// TIA Portal V15.1 export
// export: Created 2024-05-17T05:38:29.3000948Z, ExportSetting WithDefaults, DisplayName Totally Integrated Automation Portal, DisplayVersion V15.1 Update 5, DisplayName TIA Portal Openness, DisplayVersion V15.1 Update 5, DisplayName SINAMICS Startdrive Advanced, DisplayVersion V15.1, DisplayName G130, G150, S120, S150, SINAMICS MV, S210, DisplayVersion V15.1, DisplayName G110M, G120, G120C, G120D, G120P, DisplayVersion V15.1, DisplayName STEP 7 Professional, DisplayVersion V15.1 Update 5, DisplayName STEP 7 Safety, DisplayVersion V15.1, DisplayName WinCC Professional, DisplayVersion V15.1 Update 5, DisplayName SIMATIC Visualization Architect, DisplayVersion V15.1
FUNCTION_BLOCK "LETAFuseCPC20PNSub"   // FB1407, SCL
{ S7_Optimized_Access := 'TRUE' }
VERSION : 0.1
// stored: AutoNumber false, IsIECCheckEnabled false, IsRetainMemResEnabled false, MemoryReserve 100, SetENOAutomatically False, UDAEnableTagReadback false
   VAR_INPUT
      I_NewShift { ExternalAccessible := 'False'; ExternalVisible := 'False'; ExternalWritable := 'False'} : Bool;   // NewShift / Morning shift
      I_ReadNomCurr { ExternalAccessible := 'False'; ExternalVisible := 'False'; ExternalWritable := 'False'} : Bool;   // HMI Command - Read nominal current
      I_CancelReadNomCurr { ExternalAccessible := 'False'; ExternalVisible := 'False'; ExternalWritable := 'False'} : Bool;   // HMI Command - Cancel Read nominal current
      C_HWInput { ExternalAccessible := 'False'; ExternalVisible := 'False'; ExternalWritable := 'False'} : HW_IO;   // Slot ID from CPC20PN
      C_Block1_TotalCurrent { ExternalAccessible := 'False'; ExternalVisible := 'False'; ExternalWritable := 'False'} : HW_IO;   // Base Module Slot ID Total Current, 0=not in use.
      C_Block1_StatusControl { ExternalAccessible := 'False'; ExternalVisible := 'False'; ExternalWritable := 'False'} : HW_IO;   // Base Module Slot ID Status / Control, 0=not in use.
      "C_Block1_MeasurementU/I" { ExternalAccessible := 'False'; ExternalVisible := 'False'; ExternalWritable := 'False'} : HW_IO;   // Base Module Slot ID Measurement UI, 0=not in use.
      C_Block2_TotalCurrent { ExternalAccessible := 'False'; ExternalVisible := 'False'; ExternalWritable := 'False'} : HW_IO;   // Extension Module Slot ID Total Current, 0=not in use.
      C_Block2_StatusControl { ExternalAccessible := 'False'; ExternalVisible := 'False'; ExternalWritable := 'False'} : HW_IO;   // Extension Module Slot ID Status / Control, 0=not in use.
      "C_Block2_MeasurementU/I" { ExternalAccessible := 'False'; ExternalVisible := 'False'; ExternalWritable := 'False'} : HW_IO;   // Extension Module Slot ID Measurement UI, 0=not in use.
      C_Config { ExternalAccessible := 'False'; ExternalVisible := 'False'; ExternalWritable := 'False'} : "ETAFuseCPC20PNConfig";   // Config
   END_VAR
   VAR_OUTPUT
      O_StatusCPC20_Bit0 { ExternalAccessible := 'False'; ExternalVisible := 'False'; ExternalWritable := 'False'} : Bool;   // Bit0 = no configuration data available
      O_StatusCPC20_Bit1 { ExternalAccessible := 'False'; ExternalVisible := 'False'; ExternalWritable := 'False'} : Bool;   // Bit1 = invalid configuration data
      O_StatusCPC20_Bit4 { ExternalAccessible := 'False'; ExternalVisible := 'False'; ExternalWritable := 'False'} : Bool;   // Bit4 = command buffer overflow
      O_StatusCPC20_Bit7 { ExternalAccessible := 'False'; ExternalVisible := 'False'; ExternalWritable := 'False'} : Bool;   // Bit7 = no communication with at least one PWR board
      O_StatusCPC20_Bit9 { ExternalAccessible := 'False'; ExternalVisible := 'False'; ExternalWritable := 'False'} : Bool;   // Bit9 = CPC temporary error
      O_StatusCPC20_Bit10 { ExternalAccessible := 'False'; ExternalVisible := 'False'; ExternalWritable := 'False'} : Bool;   // Bit10 = CPC hardware error
      O_ReadNomCurrActive { ExternalAccessible := 'False'; ExternalVisible := 'False'; ExternalWritable := 'False'} : Bool;   // Reading of nominal current is active
      O_ReadNomCurrFuseNr { ExternalAccessible := 'False'; ExternalVisible := 'False'; ExternalWritable := 'False'} : Int;   // Fuse number Reading of nominal current
      O_AlarmReadNomCurr { ExternalAccessible := 'False'; ExternalVisible := 'False'; ExternalWritable := 'False'} : Bool;   // Overtime Reading of nominal current
      O_Block1TotalCurrent { ExternalAccessible := 'False'; ExternalVisible := 'False'; ExternalWritable := 'False'} : Real;   // Total current Block 1
      O_Block2TotalCurrent { ExternalAccessible := 'False'; ExternalVisible := 'False'; ExternalWritable := 'False'} : Real;   // Total current Block 2
   END_VAR
   VAR_IN_OUT
      IO_ETAFuseData : "ETAFuseData";   // ETA fuse status
      H_ETAFuseCPC20PN : "H_ETAFuseCPC20PN";   // Animation
   END_VAR
   VAR
      InitNominalCurrent { ExternalAccessible := 'False'; ExternalVisible := 'False'; ExternalWritable := 'False'} : Bool;   // Read once all Nominal Currents at Startup
      ChannelNumber { ExternalAccessible := 'False'; ExternalVisible := 'False'; ExternalWritable := 'False'} : Int;   // Channel Number
      Block1Size { ExternalAccessible := 'False'; ExternalVisible := 'False'; ExternalWritable := 'False'} : Int;   // Block size
      Block2Size { ExternalAccessible := 'False'; ExternalVisible := 'False'; ExternalWritable := 'False'} : Int;   // Block size
      HardwareID { ExternalAccessible := 'False'; ExternalVisible := 'False'; ExternalWritable := 'False'} : HW_IO;   // HW IO
      i { ExternalAccessible := 'False'; ExternalVisible := 'False'; ExternalWritable := 'False'} : Int;   // Loop Counter
      iCount { ExternalAccessible := 'False'; ExternalVisible := 'False'; ExternalWritable := 'False'} : Int;   // Loop Counter To Go Threw All Channels
      iCalcAddress { ExternalAccessible := 'False'; ExternalVisible := 'False'; ExternalWritable := 'False'} : Int;   // Fuse Adress To Be Calculated
      iCountGet { ExternalAccessible := 'False'; ExternalVisible := 'False'; ExternalWritable := 'False'} : Int;   // Sequence Pointer Get Data
      iCountNominalCurrent { ExternalAccessible := 'False'; ExternalVisible := 'False'; ExternalWritable := 'False'} : Int;   // Loop Counter To Go Threw All Channels
      BuildStatus { ExternalAccessible := 'False'; ExternalVisible := 'False'; ExternalWritable := 'False'} : Word;   // BuildStatus
      iError { ExternalAccessible := 'False'; ExternalVisible := 'False'; ExternalWritable := 'False'} : Int;   // iError
      CalcValue { ExternalAccessible := 'False'; ExternalVisible := 'False'; ExternalWritable := 'False'} : Int;   // CalcValue
      EmptyDataCPC20 { ExternalAccessible := 'False'; ExternalVisible := 'False'; ExternalWritable := 'False'} : Struct   // Empty struct to delete info
         Voltage { ExternalAccessible := 'False'; ExternalVisible := 'False'; ExternalWritable := 'False'} : Real;   // Voltage
         Current { ExternalAccessible := 'False'; ExternalVisible := 'False'; ExternalWritable := 'False'} : Real;   // Current
         NominalCurrent { ExternalAccessible := 'False'; ExternalVisible := 'False'; ExternalWritable := 'False'} : Byte;   // Nominal Current
         Status { ExternalAccessible := 'False'; ExternalVisible := 'False'; ExternalWritable := 'False'} : Byte;   // Status
         Control { ExternalAccessible := 'False'; ExternalVisible := 'False'; ExternalWritable := 'False'} : Byte;   // Control
      END_STRUCT;
      EmptyForHMIFuse { ExternalAccessible := 'False'; ExternalVisible := 'False'; ExternalWritable := 'False'} : Struct   // Empty struct to delete info
         Used { ExternalAccessible := 'False'; ExternalVisible := 'False'; ExternalWritable := 'False'} : Bool;   // Used
         "SwitchOn/OFFOnlyCabinet" { ExternalAccessible := 'False'; ExternalVisible := 'False'; ExternalWritable := 'False'} : Bool;   // Switch On/Off only posible in the cabinet, button on the fuse
         IAnim { ExternalAccessible := 'False'; ExternalVisible := 'False'; ExternalWritable := 'False'} : Word;   // IAnim
         Status { ExternalAccessible := 'False'; ExternalVisible := 'False'; ExternalWritable := 'False'} : Byte;   // Status
         AlarmActive { ExternalAccessible := 'False'; ExternalVisible := 'False'; ExternalWritable := 'False'} : Bool;   // Alarm Active
      END_STRUCT;
      EmptyForHMIChannelInfo { ExternalAccessible := 'False'; ExternalVisible := 'False'; ExternalWritable := 'False'} : Struct   // Empty struct to delete info
         "Name" { ExternalAccessible := 'False'; ExternalVisible := 'False'; ExternalWritable := 'False'} : String[40];   // Fuse name
         Description { ExternalAccessible := 'False'; ExternalVisible := 'False'; ExternalWritable := 'False'} : String[60];   // Description
         Current { ExternalAccessible := 'False'; ExternalVisible := 'False'; ExternalWritable := 'False'} : Real;   // Current
         NominalCurrent { ExternalAccessible := 'False'; ExternalVisible := 'False'; ExternalWritable := 'False'} : Int;   // Nominal Current
      END_STRUCT;
      NonCyclicCommunication { ExternalAccessible := 'False'; ExternalVisible := 'False'; ExternalWritable := 'False'} : Struct   // Non cyclic communication variables
         H_ReadNomCurrTrig { ExternalAccessible := 'False'; ExternalVisible := 'False'; ExternalWritable := 'False'} : Bool;   // HMI button to start reading nominal current
         ReadNomCurrActive { ExternalAccessible := 'False'; ExternalVisible := 'False'; ExternalWritable := 'False'} : Bool;   // Reading of nominal current is active
      END_STRUCT;
      Get { ExternalAccessible := 'False'; ExternalVisible := 'False'; ExternalWritable := 'False'} : Struct   // FB
         bGetData { ExternalAccessible := 'False'; ExternalVisible := 'False'; ExternalWritable := 'False'} : Bool;
         bValid { ExternalAccessible := 'False'; ExternalVisible := 'False'; ExternalWritable := 'False'} : Bool;
         bBusy { ExternalAccessible := 'False'; ExternalVisible := 'False'; ExternalWritable := 'False'} : Bool;
         diIndex { ExternalAccessible := 'False'; ExternalVisible := 'False'; ExternalWritable := 'False'} : DInt;
         uiMlen { ExternalAccessible := 'False'; ExternalVisible := 'False'; ExternalWritable := 'False'} : UInt;
         uilen { ExternalAccessible := 'False'; ExternalVisible := 'False'; ExternalWritable := 'False'} : UInt;
         bError { ExternalAccessible := 'False'; ExternalVisible := 'False'; ExternalWritable := 'False'} : Bool;
         dwState { ExternalAccessible := 'False'; ExternalVisible := 'False'; ExternalWritable := 'False'} : DWord;
         TonError { ExternalAccessible := 'False'; ExternalVisible := 'False'; ExternalWritable := 'False'} : Bool;
         DataByte { ExternalAccessible := 'False'; ExternalVisible := 'False'; ExternalWritable := 'False'} : Array[1..20] of Byte;
      END_STRUCT;
      RDREC_FB { ExternalAccessible := 'False'; ExternalVisible := 'False'; ExternalWritable := 'False'} : RDREC;   // FB
      StatusCPC20 { ExternalAccessible := 'False'; ExternalVisible := 'False'; ExternalWritable := 'False'} : Array[0..1] of Byte;   // Temp
      Current { ExternalAccessible := 'False'; ExternalVisible := 'False'; ExternalWritable := 'False'} : Array[0..1] of Byte;   // Temp
      Status { ExternalAccessible := 'False'; ExternalVisible := 'False'; ExternalWritable := 'False'} : Array[1..32] of Byte;   // Temp
      Control { ExternalAccessible := 'False'; ExternalVisible := 'False'; ExternalWritable := 'False'} : Array[1..32] of Byte;   // Temp
      UI { ExternalAccessible := 'False'; ExternalVisible := 'False'; ExternalWritable := 'False'} : Array[0..130] of Byte;   // Temp
      T_ReadNomCurr { ExternalAccessible := 'False'; ExternalVisible := 'False'; ExternalWritable := 'False'} : TON_TIME;   // Timer
   END_VAR
BEGIN
   (*=================================================================================*)
   (* Init at startup *)
   (*=================================================================================*)
   IF "FirstScan" THEN
       #InitNominalCurrent := True;
   END_IF;

   (*=================================================================================*)
   (* Check number of protectors active *)
   (*=================================================================================*)
   #Block1Size := 0;
   IF #C_Config.Fuse[1].Used THEN
       #Block1Size := 1;
   END_IF;
   IF #C_Config.Fuse[3].Used THEN
       #Block1Size := 2;
   END_IF;
   IF #C_Config.Fuse[5].Used THEN
       #Block1Size := 3;
   END_IF;
   IF #C_Config.Fuse[7].Used THEN
       #Block1Size := 4;
   END_IF;
   IF #C_Config.Fuse[9].Used THEN
       #Block1Size := 5;
   END_IF;
   IF #C_Config.Fuse[11].Used THEN
       #Block1Size := 6;
   END_IF;
   IF #C_Config.Fuse[13].Used THEN
       #Block1Size := 7;
   END_IF;
   IF #C_Config.Fuse[15].Used THEN
       #Block1Size := 8;
   END_IF;
   IF #C_Config.Fuse[17].Used THEN
       #Block1Size := 9;
   END_IF;
   IF #C_Config.Fuse[19].Used THEN
       #Block1Size := 10;
   END_IF;
   IF #C_Config.Fuse[21].Used THEN
       #Block1Size := 11;
   END_IF;
   IF #C_Config.Fuse[23].Used THEN
       #Block1Size := 12;
   END_IF;
   IF #C_Config.Fuse[25].Used THEN
       #Block1Size := 13;
   END_IF;
   IF #C_Config.Fuse[27].Used THEN
       #Block1Size := 14;
   END_IF;
   IF #C_Config.Fuse[29].Used THEN
       #Block1Size := 15;
   END_IF;
   IF #C_Config.Fuse[31].Used THEN
       #Block1Size := 16;
   END_IF;

   #Block2Size := 0;
   IF #C_Config.Fuse[33].Used THEN
       #Block2Size := 1;
   END_IF;
   IF #C_Config.Fuse[35].Used THEN
       #Block2Size :=2;
   END_IF;
   IF #C_Config.Fuse[37].Used THEN
       #Block2Size := 3;
   END_IF;
   IF #C_Config.Fuse[39].Used THEN
       #Block2Size := 4;
   END_IF;
   IF #C_Config.Fuse[41].Used THEN
       #Block2Size := 5;
   END_IF;
   IF #C_Config.Fuse[43].Used THEN
       #Block2Size := 6;
   END_IF;
   IF #C_Config.Fuse[45].Used THEN
       #Block2Size := 7;
   END_IF;
   IF #C_Config.Fuse[47].Used THEN
       #Block2Size := 8;
   END_IF;
   IF #C_Config.Fuse[49].Used THEN
       #Block2Size := 9;
   END_IF;
   IF #C_Config.Fuse[51].Used THEN
       #Block2Size := 10;
   END_IF;
   IF #C_Config.Fuse[53].Used THEN
       #Block2Size := 11;
   END_IF;
   IF #C_Config.Fuse[55].Used THEN
       #Block2Size := 12;
   END_IF;
   IF #C_Config.Fuse[57].Used THEN
       #Block2Size := 13;
   END_IF;
   IF #C_Config.Fuse[59].Used THEN
       #Block2Size := 14;
   END_IF;
   IF #C_Config.Fuse[61].Used THEN
       #Block2Size := 15;
   END_IF;
   IF #C_Config.Fuse[63].Used THEN
       #Block2Size := 16;
   END_IF;

   (*=================================================================================*)
   (* CPC20   ---   Read State *)
   (*=================================================================================*)
   IF #C_HWInput > 0 THEN
       (*Read Data*)
       #iError := DPRD_DAT(LADDR := #C_HWInput, RECORD => #StatusCPC20);
       (*Calculate Value*)
       #BuildStatus := #StatusCPC20[0];
       #BuildStatus := SHL(IN := #BuildStatus, N := 8);
   END_IF;

   #O_StatusCPC20_Bit0 := #BuildStatus.%X0;
   #O_StatusCPC20_Bit1 := #BuildStatus.%X1;
   #O_StatusCPC20_Bit4 := #BuildStatus.%X4;
   #O_StatusCPC20_Bit7 := #BuildStatus.%X7;
   #O_StatusCPC20_Bit9 := #BuildStatus.%X9;
   #O_StatusCPC20_Bit10 := #BuildStatus.%X10;

   (*=================================================================================*)
   (* AM03_1   ---   Read Status + Send Control / Read Voltage + Current *)
   (*=================================================================================*)
   IF #Block1Size > 0 THEN
       // Read Total current and calculate it
       IF #C_Block1_TotalCurrent > 0 THEN
           (*Read Data*)
           #iError := DPRD_DAT(LADDR := #C_Block1_TotalCurrent, RECORD => #Current);
           (*Calculate Value*)
           #CalcValue := #Current[1];
           #CalcValue := SHL(IN := #CalcValue, N := 8);
           #O_Block1TotalCurrent := (#CalcValue + #Current[0]) / 100;
       END_IF;
       (*Status and Control*)
       IF #C_Block1_StatusControl > 0 THEN
           (*Read Inputs*)
           #iError := DPRD_DAT(LADDR := #C_Block1_StatusControl, RECORD => #Status);
           (*Take it over to the Datastructure*)
           FOR #iCount := 1 TO 32 DO
               IF #iCount <= #Block1Size * 2 THEN
                   IF "SimulationActive" THEN
                       "NotUsedBool" := False;
                     ELSE
                       #IO_ETAFuseData.DataCPC20.Fuse[#iCount].Status := #Status[#iCount]; (*Read Status*)
                   END_IF;
                   #Control[#iCount] := #IO_ETAFuseData.DataCPC20.Fuse[#iCount].Control ; (*Write control to the buffer*)
               ELSE
                   #IO_ETAFuseData.DataCPC20.Fuse[#iCount].Status := 255; (*Read Status*)
                   #Control[#iCount] := 0; (*Write control to the buffer*)
               END_IF;
           END_FOR;
           (*Write outputs to the CPC*)
           #iError := DPWR_DAT(LADDR := #C_Block1_StatusControl, RECORD := #Control);
       END_IF;
       (*Measurement preperation*)
       IF #"C_Block1_MeasurementU/I" > 0 THEN
           (*Read measurenets values*)
           #iError := DPRD_DAT(LADDR := #"C_Block1_MeasurementU/I", RECORD => #UI);
           (*Create Measurements*)
           FOR #iCount := 1 TO 32 DO
               (*Calculate new Adress*)
               #iCalcAddress := ((#iCount - 1) * 4);
               IF #iCount <= #Block1Size * 2 THEN
                   (*Calculate current and take it over to the Datastructure*)
                   #CalcValue := #UI[#iCalcAddress + 1]; (*-2*)
                   #CalcValue := SHL(IN := #CalcValue, N := 8);
                   #IO_ETAFuseData.DataCPC20.Fuse[#iCount].Current := INT_TO_REAL(#CalcValue + #UI[#iCalcAddress]) / 100; (*-3*)
                   (*Calculate voltage and take it over to the Datastructure*)
                   #CalcValue := #UI[#iCalcAddress + 3];
                   #CalcValue := SHL(IN := #CalcValue, N := 8); (*-0*)
                   #IO_ETAFuseData.DataCPC20.Fuse[#iCount].Voltage := INT_TO_REAL(#CalcValue + #UI[#iCalcAddress + 2]) / 100; (*-1*)
               ELSE
                   #IO_ETAFuseData.DataCPC20.Fuse[#iCount].Current := 0; (*-3*)
                   #IO_ETAFuseData.DataCPC20.Fuse[#iCount].Voltage := 0; (*-1*)
               END_IF;
           END_FOR;
       END_IF;
   END_IF;

   (*=================================================================================*)
   (* AM03_2   ---   Read Status + Send Control / Read Voltage + Current *)
   (*=================================================================================*)
   IF #Block2Size > 0 THEN
       // Read Total current and calculate it
       IF #C_Block2_TotalCurrent > 0 THEN
           (*Read Data*)
           #iError := DPRD_DAT(LADDR := #C_Block2_TotalCurrent, RECORD => #Current);
           (*Calculate Value*)
           #CalcValue := #Current[1];
           #CalcValue := SHL(IN := #CalcValue, N := 8);
           #O_Block2TotalCurrent := (#CalcValue + #Current[0]) / 100;
       END_IF;
       (*Status And Control*)
       IF #C_Block2_StatusControl > 0 THEN
           (*Read Inputs*)
           #iError := DPRD_DAT(LADDR := #C_Block2_StatusControl, RECORD => #Status);
           (*Take it over to the Datastructure*)
           FOR #iCount := 1 TO 32 DO
               IF #iCount <= #Block2Size * 2 THEN //WDL changed C_Block1Size by C_Block2Size
                   IF "SimulationActive" THEN
                       "NotUsedBool" := False;
                     ELSE
                       #IO_ETAFuseData.DataCPC20.Fuse[#iCount + 32].Status := #Status[#iCount]; (*Read Status*)
                   END_IF;
                   #Control[#iCount] := #IO_ETAFuseData.DataCPC20.Fuse[#iCount + 32].Control; (*Write control to the buffer*)
               ELSE
                   #IO_ETAFuseData.DataCPC20.Fuse[#iCount + 32].Status := 255; (*Read Status*)
                   #Control[#iCount] := 0; (*Write control to the buffer*)
               END_IF;
           END_FOR;
           (*Write outputs to the CPC*)
           #iError := DPWR_DAT(LADDR := #C_Block2_StatusControl, RECORD := #Control);
       END_IF;
       (*Measurement preperation*)
       IF #"C_Block2_MeasurementU/I" > 0 THEN
           (*Read measurenets values*)
           #iError := DPRD_DAT(LADDR := #"C_Block2_MeasurementU/I", RECORD => #UI);
           (*Create Measurements*)
           FOR #iCount := 1 TO 32 DO
               (*Calculate new Adress*)
               #iCalcAddress := ((#iCount - 1) * 4);
               IF #iCount <= #Block2Size * 2 THEN
                   (*Calculate current and take it over to the Datastructure*)
                   #CalcValue := #UI[#iCalcAddress + 1]; (*-2*)
                   #CalcValue := SHL(IN := #CalcValue, N := 8);
                   #IO_ETAFuseData.DataCPC20.Fuse[#iCount + 32].Current := INT_TO_REAL(#CalcValue + #UI[#iCalcAddress]) / 100; (*-3*)
                   (*Calculate voltage and take it over to the Datastructure*)
                   #CalcValue := #UI[#iCalcAddress + 3];
                   #CalcValue := SHL(IN := #CalcValue, N := 8); (*-0*)
                   #IO_ETAFuseData.DataCPC20.Fuse[#iCount + 32].Voltage := INT_TO_REAL(#CalcValue + #UI[#iCalcAddress + 2]) / 100; (*-1*)
               ELSE
                   #IO_ETAFuseData.DataCPC20.Fuse[#iCount + 32].Current := 0; (*-3*)
                   #IO_ETAFuseData.DataCPC20.Fuse[#iCount + 32].Voltage := 0; (*-1*)
               END_IF;
           END_FOR;
       END_IF;
   END_IF;

   (*=================================================================================*)
   (*AM03_1 & AM03_2   ---   Read Nominal Current *)    
   (*=================================================================================*)
   //HMI Command - Cancel Read nominal current
   IF #I_CancelReadNomCurr OR "SimulationActive" THEN
       #iCountGet := 1000;
   END_IF;

   CASE #iCountGet OF
       0: IF (#InitNominalCurrent OR #I_ReadNomCurr OR #I_NewShift) AND NOT #NonCyclicCommunication.ReadNomCurrActive AND NOT "SimulationActive" THEN
               IF (#C_Block1_TotalCurrent > 0) THEN
                   #iCountNominalCurrent := 1; // Init Value
                   #ChannelNumber := 1; // Init Value
                   #HardwareID := #C_Block1_TotalCurrent; // Init Value
                   #NonCyclicCommunication.ReadNomCurrActive := True;
                   #iCountGet := 10;
               END_IF;

               IF (#C_Block1_TotalCurrent = 0) AND (#C_Block2_TotalCurrent > 0) THEN
                   #iCountNominalCurrent := 33; // Init Value
                   #ChannelNumber := 1; // Init Value
                   #HardwareID := #C_Block2_TotalCurrent; // Init Value
                   #NonCyclicCommunication.ReadNomCurrActive := True;
                   #iCountGet := 10;
               END_IF;

               IF (#C_Block1_TotalCurrent = 0) AND (#C_Block2_TotalCurrent = 0) THEN
                   #Get.bGetData := False;
                   #iCountGet := 1000;
               END_IF;
           END_IF;
       10: // Set Parameter to read a channel and start it
           IF NOT #C_Config.Fuse[#iCountNominalCurrent].Used THEN
               #iCountNominalCurrent := #iCountNominalCurrent + 1;
               #ChannelNumber := #ChannelNumber + 1;
               #IO_ETAFuseData.DataCPC20.Fuse[#iCountNominalCurrent].NominalCurrent := 0;
               #iCountGet := 100;
           ELSE
               #Get.diIndex := (#ChannelNumber * 100) + 1; // Channel Number * Factor for Parameter + Index
               #Get.uiMlen := 8;
               #Get.bGetData := True; (*Read Data*)
               #iCountGet := 20;
           END_IF;

           IF (#iCountNominalCurrent >= 64) THEN
               #iCountGet := 1000;
           END_IF;
       20: (*reading is active*)
           IF #Get.bBusy OR #Get.bError THEN
               #Get.bGetData := false; (*Edge to read is enough*)
               #iCountGet := 30;
           END_IF;
       30: (*Evaluate data, stop reading, set message in case of error*)
           IF NOT #Get.bBusy THEN
               IF #Get.bValid THEN
                   #IO_ETAFuseData.DataCPC20.Fuse[#iCountNominalCurrent].NominalCurrent := #Get.DataByte[1] - 16#A0;
                   #iCountGet := 100;
               ELSE
                   #iCountGet := 10;
               END_IF;
           END_IF;
       100: // check for next channel
           IF (#iCountNominalCurrent >= 32) AND (#iCountNominalCurrent < 64) THEN
               #HardwareID := #C_Block2_TotalCurrent;
               #iCountNominalCurrent := #iCountNominalCurrent + 1;
               #ChannelNumber := #ChannelNumber + 1;
               #iCountGet := 10;
           END_IF;

           IF #iCountNominalCurrent < 32 THEN
               #HardwareID := #C_Block1_TotalCurrent;
               #iCountNominalCurrent := #iCountNominalCurrent + 1;
               #ChannelNumber := #ChannelNumber + 1;
               #iCountGet := 10;
           END_IF;

           IF (#iCountNominalCurrent = 33) THEN
               #ChannelNumber := 1;
           END_IF;

           IF (#iCountNominalCurrent >= 64) THEN
               #iCountGet := 1000;
           END_IF;
       1000: // End
           #InitNominalCurrent := False;
           #NonCyclicCommunication.ReadNomCurrActive := False;
           #iCountGet := 0;
   END_CASE;

   // Reading of nominal current is active
   #O_ReadNomCurrActive := #NonCyclicCommunication.ReadNomCurrActive;
   #O_ReadNomCurrFuseNr := #iCountNominalCurrent;

   // Overtime Reading of nominal current
   #T_ReadNomCurr(IN:= #O_ReadNomCurrActive,
                  PT:= T#60s);

   #O_AlarmReadNomCurr := #T_ReadNomCurr.Q;

   // Call noncyclic communication
   #RDREC_FB(REQ := #Get.bGetData,
             ID := #HardwareID,
             INDEX := #Get.diIndex,
             MLEN := #Get.uiMlen,
             VALID => #Get.bValid,
             BUSY => #Get.bBusy,
             ERROR => #Get.bError,
             STATUS => #Get.dwState,
             LEN => #Get.uilen,
             RECORD := #Get.DataByte);

   (*=================================================================================*)
   (* Fill-in/Clear Information *)    
   (*=================================================================================*)
   FOR #iCount := 1 TO 64 DO
       IF #C_Config.Fuse[#iCount].Used THEN
           #IO_ETAFuseData.ForHMICPC20.Fuse[#iCount].Used := True;
           #H_ETAFuseCPC20PN.H_ForHMI.ChannelInfo[#iCount].Name := #C_Config.Fuse[#iCount].Name;
           #H_ETAFuseCPC20PN.H_ForHMI.ChannelInfo[#iCount].Description := #C_Config.Fuse[#iCount].Description;
           #H_ETAFuseCPC20PN.H_ForHMI.ChannelInfo[#iCount].Current := #IO_ETAFuseData.DataCPC20.Fuse[#iCount].Current;
           #H_ETAFuseCPC20PN.H_ForHMI.ChannelInfo[#iCount].NominalCurrent := #IO_ETAFuseData.DataCPC20.Fuse[#iCount].NominalCurrent;
       ELSE
           #IO_ETAFuseData.DataCPC20.Fuse[#iCount] := #EmptyDataCPC20;
           #IO_ETAFuseData.DataCPC20.Fuse[#iCount].Status := 255;

           #IO_ETAFuseData.ForHMICPC20.Fuse[#iCount] := #EmptyForHMIFuse;

           #H_ETAFuseCPC20PN.H_ForHMI.Fuse[#iCount] := #EmptyForHMIFuse;
           #H_ETAFuseCPC20PN.H_ForHMI.ChannelInfo[#iCount] := #EmptyForHMIChannelInfo;
           #H_ETAFuseCPC20PN.H_ForHMI.ChannelInfo[#iCount].Name := 'Not exist';
       END_IF;
   END_FOR;

   #H_ETAFuseCPC20PN.H_ForHMI.Fuse := #IO_ETAFuseData.ForHMICPC20.Fuse;
END_FUNCTION_BLOCK
